// TIA Portal V20 export
FUNCTION "CallDiagnostic" : Void   // FC16, LAD
TITLE = Diagnostics
AUTHOR : SICAR
FAMILY : Diag
// Call of SICAR Diagnostic blocks
// stored: IsIECCheckEnabled true, SetENOAutomatically true
   VAR_TEMP
      statWStringName : WString[24];
      tempHardwareOKexample : Bool;   // REPLACE: This output can be used as an interlock for Control Modules
   END_VAR
   VAR CONSTANT
      TRUE : Bool := TRUE;
   END_VAR
   // Ret_Val : Ret_Val
   VAR_TEMP   // added for the SCL form of the ladder/FBD networks
      _w1 : Bool;
   END_VAR
BEGIN

REGION Network 1: BLOCK INFO HEADER
   // SIEMENS AG / (c)Copyright 2023
   // ------------------------------------------------------------------------------
   // Title:            CallDiagnostic (FC16)
   // Comment/Function: Call of SICAR Diagnostic blocks
   // Library/Family:   Diag
   // Author:           SICAR
   // Tested with:      ---
   // Engineering:      TIA Portal V19
   // Restrictions:     -
   // Requirements:     ---
   // ------------------------------------------------------------------------------
   // Change log table:
   // Version | Date | Expert in charge | Changes applied
   // -------|---------|-------------|--------------------------------------------
   // 01.00.00 | 01.01.1999 | Person x | First released version
   // 01.00.01 | 02.01.1999 | Person y | Block was Updated
END_REGION

REGION Network 2: Call: Diagnostic Profinet Devices
   // For diagnose the whole profinet devices of this PLC
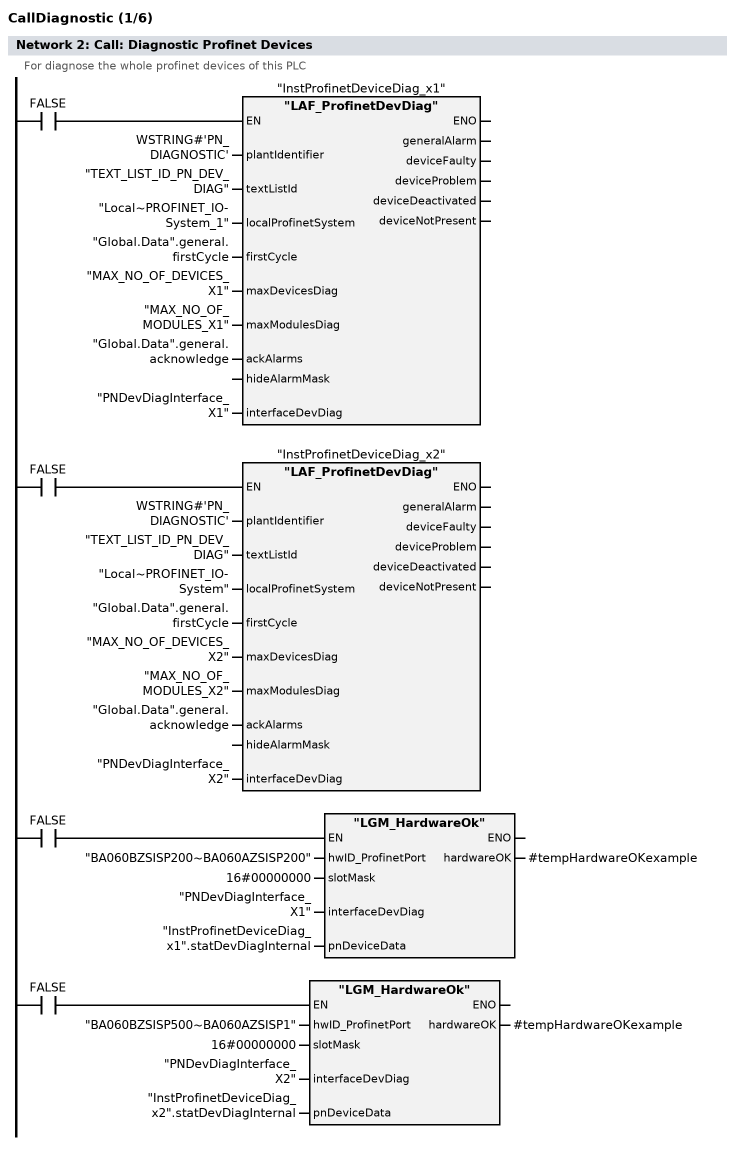
   RUNG wire#powerrail
      Contact( FALSE )
      "InstProfinetDeviceDiag_x1"(plantIdentifier := WSTRING#'PN_DIAGNOSTIC', textListId := "TEXT_LIST_ID_PN_DEV_DIAG", localProfinetSystem := "Local~PROFINET_IO-System_1", firstCycle := "Global.Data".general.firstCycle, maxDevicesDiag := "MAX_NO_OF_DEVICES_X1", maxModulesDiag := "MAX_NO_OF_MODULES_X1", ackAlarms := "Global.Data".general.acknowledge, hideAlarmMask :=, interfaceDevDiag := "PNDevDiagInterface_X1", generalAlarm =>, deviceFaulty =>, deviceProblem =>, deviceDeactivated =>, deviceNotPresent =>)
   END_RUNG
   RUNG wire#powerrail
      Contact( FALSE )
      "InstProfinetDeviceDiag_x2"(plantIdentifier := WSTRING#'PN_DIAGNOSTIC', textListId := "TEXT_LIST_ID_PN_DEV_DIAG", localProfinetSystem := "Local~PROFINET_IO-System", firstCycle := "Global.Data".general.firstCycle, maxDevicesDiag := "MAX_NO_OF_DEVICES_X2", maxModulesDiag := "MAX_NO_OF_MODULES_X2", ackAlarms := "Global.Data".general.acknowledge, hideAlarmMask :=, interfaceDevDiag := "PNDevDiagInterface_X2", generalAlarm =>, deviceFaulty =>, deviceProblem =>, deviceDeactivated =>, deviceNotPresent =>)
   END_RUNG
   RUNG wire#powerrail
      Contact( FALSE )
      "LGM_HardwareOk"(hwID_ProfinetPort := "BA060BZSISP200~BA060AZSISP200", slotMask := 16#00000000, interfaceDevDiag := "PNDevDiagInterface_X1", pnDeviceData := "InstProfinetDeviceDiag_x1".statDevDiagInternal, hardwareOK => #tempHardwareOKexample)
   END_RUNG
   RUNG wire#powerrail
      Contact( FALSE )
      "LGM_HardwareOk"(hwID_ProfinetPort := "BA060BZSISP500~BA060AZSISP1", slotMask := 16#00000000, interfaceDevDiag := "PNDevDiagInterface_X2", pnDeviceData := "InstProfinetDeviceDiag_x2".statDevDiagInternal, hardwareOK => #tempHardwareOKexample)
   END_RUNG
   // the same network as SCL:
   IF FALSE THEN
       "InstProfinetDeviceDiag_x1"(plantIdentifier := WSTRING#'PN_DIAGNOSTIC',   // "LAF_ProfinetDevDiag"
                               textListId := "TEXT_LIST_ID_PN_DEV_DIAG",
                               localProfinetSystem := "Local~PROFINET_IO-System_1",
                               firstCycle := "Global.Data".general.firstCycle,
                               maxDevicesDiag := "MAX_NO_OF_DEVICES_X1",
                               maxModulesDiag := "MAX_NO_OF_MODULES_X1",
                               ackAlarms := "Global.Data".general.acknowledge,
                               interfaceDevDiag := "PNDevDiagInterface_X1");
       "InstProfinetDeviceDiag_x2"(plantIdentifier := WSTRING#'PN_DIAGNOSTIC',   // "LAF_ProfinetDevDiag"
                               textListId := "TEXT_LIST_ID_PN_DEV_DIAG",
                               localProfinetSystem := "Local~PROFINET_IO-System",
                               firstCycle := "Global.Data".general.firstCycle,
                               maxDevicesDiag := "MAX_NO_OF_DEVICES_X2",
                               maxModulesDiag := "MAX_NO_OF_MODULES_X2",
                               ackAlarms := "Global.Data".general.acknowledge,
                               interfaceDevDiag := "PNDevDiagInterface_X2");
       "LGM_HardwareOk"(hwID_ProfinetPort := "BA060BZSISP200~BA060AZSISP200",
                        slotMask := 16#00000000,
                        interfaceDevDiag := "PNDevDiagInterface_X1",
                        pnDeviceData := "InstProfinetDeviceDiag_x1".statDevDiagInternal,
                        hardwareOK => #tempHardwareOKexample);
       "LGM_HardwareOk"(hwID_ProfinetPort := "BA060BZSISP500~BA060AZSISP1",
                        slotMask := 16#00000000,
                        interfaceDevDiag := "PNDevDiagInterface_X2",
                        pnDeviceData := "InstProfinetDeviceDiag_x2".statDevDiagInternal,
                        hardwareOK => #tempHardwareOKexample);
   END_IF;
END_REGION

REGION Network 3: Call: Diagnostic Bool Interface Signals
   // Call the interface bool blocks to show boolean signals on the HMI
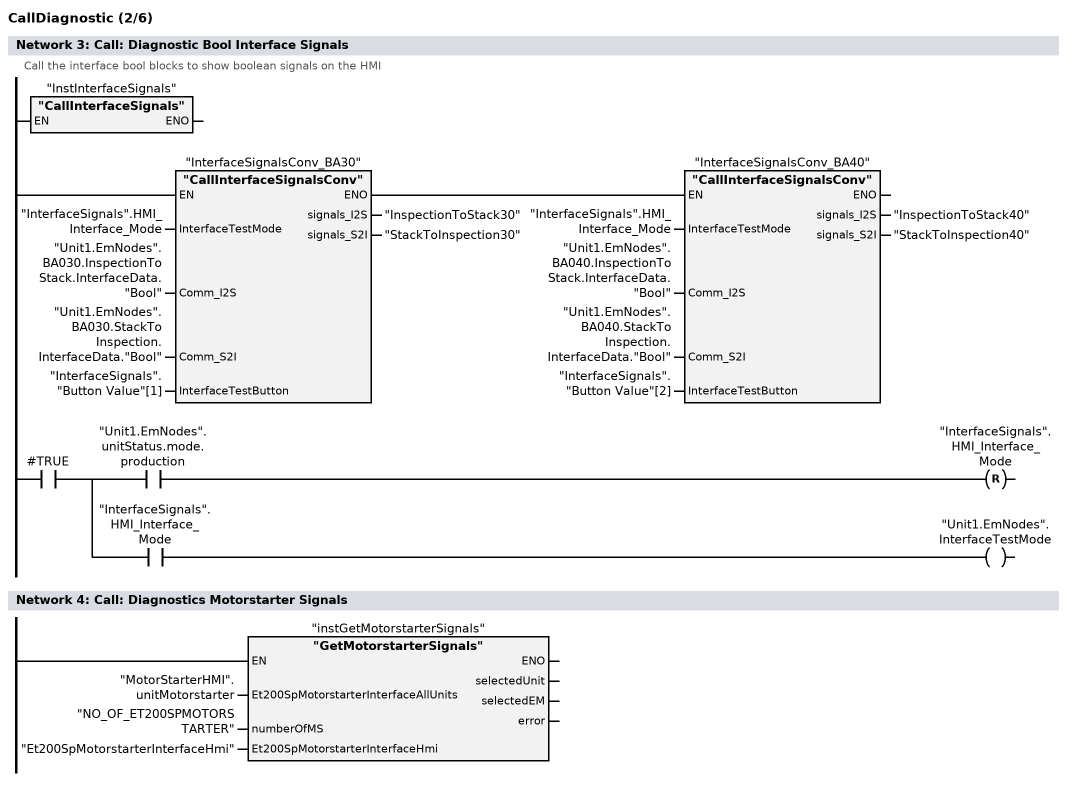
   RUNG wire#powerrail
      "InstInterfaceSignals"()
   END_RUNG
   RUNG wire#powerrail
      "InterfaceSignalsConv_BA30"(InterfaceTestMode := "InterfaceSignals".HMI_Interface_Mode, Comm_I2S := "Unit1.EmNodes".BA030.InspectionToStack.InterfaceData."Bool", Comm_S2I := "Unit1.EmNodes".BA030.StackToInspection.InterfaceData."Bool", InterfaceTestButton := "InterfaceSignals"."Button Value"[1], signals_I2S => "InspectionToStack30", signals_S2I => "StackToInspection30")
      "InterfaceSignalsConv_BA40"(InterfaceTestMode := "InterfaceSignals".HMI_Interface_Mode, Comm_I2S := "Unit1.EmNodes".BA040.InspectionToStack.InterfaceData."Bool", Comm_S2I := "Unit1.EmNodes".BA040.StackToInspection.InterfaceData."Bool", InterfaceTestButton := "InterfaceSignals"."Button Value"[2], signals_I2S => "InspectionToStack40", signals_S2I => "StackToInspection40")
   END_RUNG
   RUNG wire#powerrail
      Contact( #TRUE )
      wire#w1
      Contact( "Unit1.EmNodes".unitStatus.mode.production )
      R_Coil( "InterfaceSignals".HMI_Interface_Mode )
   END_RUNG
   RUNG wire#w1
      Contact( "InterfaceSignals".HMI_Interface_Mode )
      Coil( "Unit1.EmNodes".InterfaceTestMode )
   END_RUNG
   // the same network as SCL:
   "InstInterfaceSignals"();   // "CallInterfaceSignals"
   "InterfaceSignalsConv_BA30"(InterfaceTestMode := "InterfaceSignals".HMI_Interface_Mode,   // "CallInterfaceSignalsConv"
                           Comm_I2S := "Unit1.EmNodes".BA030.InspectionToStack.InterfaceData."Bool",
                           Comm_S2I := "Unit1.EmNodes".BA030.StackToInspection.InterfaceData."Bool",
                           InterfaceTestButton := "InterfaceSignals"."Button Value"[1],
                           signals_I2S => "InspectionToStack30",
                           signals_S2I => "StackToInspection30",
                           ENO => #_w1);
   IF #_w1 THEN
       "InterfaceSignalsConv_BA40"(InterfaceTestMode := "InterfaceSignals".HMI_Interface_Mode,   // "CallInterfaceSignalsConv"
                               Comm_I2S := "Unit1.EmNodes".BA040.InspectionToStack.InterfaceData."Bool",
                               Comm_S2I := "Unit1.EmNodes".BA040.StackToInspection.InterfaceData."Bool",
                               InterfaceTestButton := "InterfaceSignals"."Button Value"[2],
                               signals_I2S => "InspectionToStack40",
                               signals_S2I => "StackToInspection40");
   END_IF;
   IF #TRUE AND "Unit1.EmNodes".unitStatus.mode.production THEN
       "InterfaceSignals".HMI_Interface_Mode := FALSE;
   END_IF;
   "Unit1.EmNodes".InterfaceTestMode := #TRUE AND "InterfaceSignals".HMI_Interface_Mode;
END_REGION

REGION Network 4: Call: Diagnostics Motorstarter Signals
   RUNG wire#powerrail
      "instGetMotorstarterSignals"(Et200SpMotorstarterInterfaceAllUnits := "MotorStarterHMI".unitMotorstarter, numberOfMS := "NO_OF_ET200SPMOTORSTARTER", Et200SpMotorstarterInterfaceHmi := "Et200SpMotorstarterInterfaceHmi", selectedUnit =>, selectedEM =>, error =>)
   END_RUNG
   // the same network as SCL:
   "instGetMotorstarterSignals"(Et200SpMotorstarterInterfaceAllUnits := "MotorStarterHMI".unitMotorstarter,   // "GetMotorstarterSignals"
                           numberOfMS := "NO_OF_ET200SPMOTORSTARTER",
                           Et200SpMotorstarterInterfaceHmi := "Et200SpMotorstarterInterfaceHmi");
END_REGION

REGION Network 5: Call: Diagnostics Drives
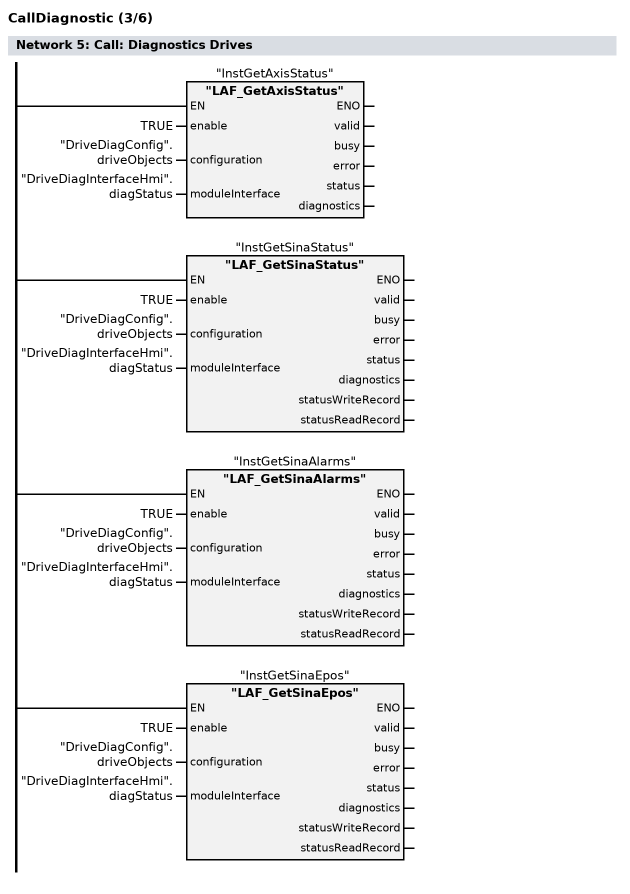
   RUNG wire#powerrail
      "InstGetAxisStatus"(enable := TRUE, configuration := "DriveDiagConfig".driveObjects, moduleInterface := "DriveDiagInterfaceHmi".diagStatus, valid =>, busy =>, error =>, status =>, diagnostics =>)
   END_RUNG
   RUNG wire#powerrail
      "InstGetSinaStatus"(enable := TRUE, configuration := "DriveDiagConfig".driveObjects, moduleInterface := "DriveDiagInterfaceHmi".diagStatus, valid =>, busy =>, error =>, status =>, diagnostics =>, statusWriteRecord =>, statusReadRecord =>)
   END_RUNG
   RUNG wire#powerrail
      "InstGetSinaAlarms"(enable := TRUE, configuration := "DriveDiagConfig".driveObjects, moduleInterface := "DriveDiagInterfaceHmi".diagStatus, valid =>, busy =>, error =>, status =>, diagnostics =>, statusWriteRecord =>, statusReadRecord =>)
   END_RUNG
   RUNG wire#powerrail
      "InstGetSinaEpos"(enable := TRUE, configuration := "DriveDiagConfig".driveObjects, moduleInterface := "DriveDiagInterfaceHmi".diagStatus, valid =>, busy =>, error =>, status =>, diagnostics =>, statusWriteRecord =>, statusReadRecord =>)
   END_RUNG
   // the same network as SCL:
   "InstGetAxisStatus"(enable := TRUE,   // "LAF_GetAxisStatus"
                       configuration := "DriveDiagConfig".driveObjects,
                       moduleInterface := "DriveDiagInterfaceHmi".diagStatus);
   "InstGetSinaStatus"(enable := TRUE,   // "LAF_GetSinaStatus"
                       configuration := "DriveDiagConfig".driveObjects,
                       moduleInterface := "DriveDiagInterfaceHmi".diagStatus);
   "InstGetSinaAlarms"(enable := TRUE,   // "LAF_GetSinaAlarms"
                       configuration := "DriveDiagConfig".driveObjects,
                       moduleInterface := "DriveDiagInterfaceHmi".diagStatus);
   "InstGetSinaEpos"(enable := TRUE,   // "LAF_GetSinaEpos"
                     configuration := "DriveDiagConfig".driveObjects,
                     moduleInterface := "DriveDiagInterfaceHmi".diagStatus);
END_REGION

REGION Network 6: Call: Servo Torque Cal (DR1~10)
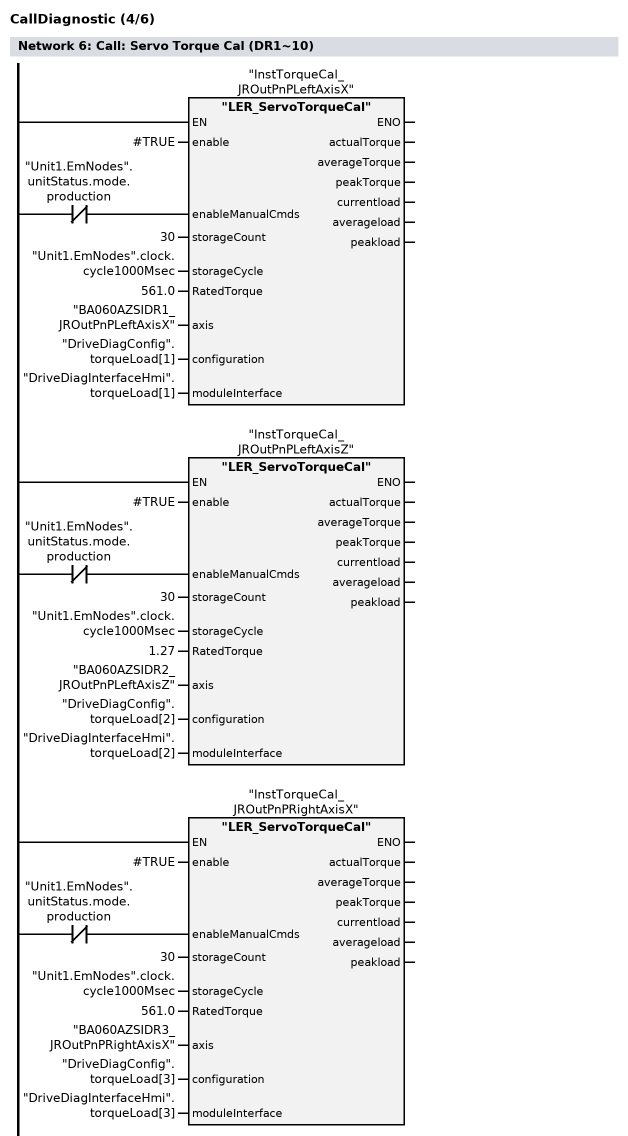
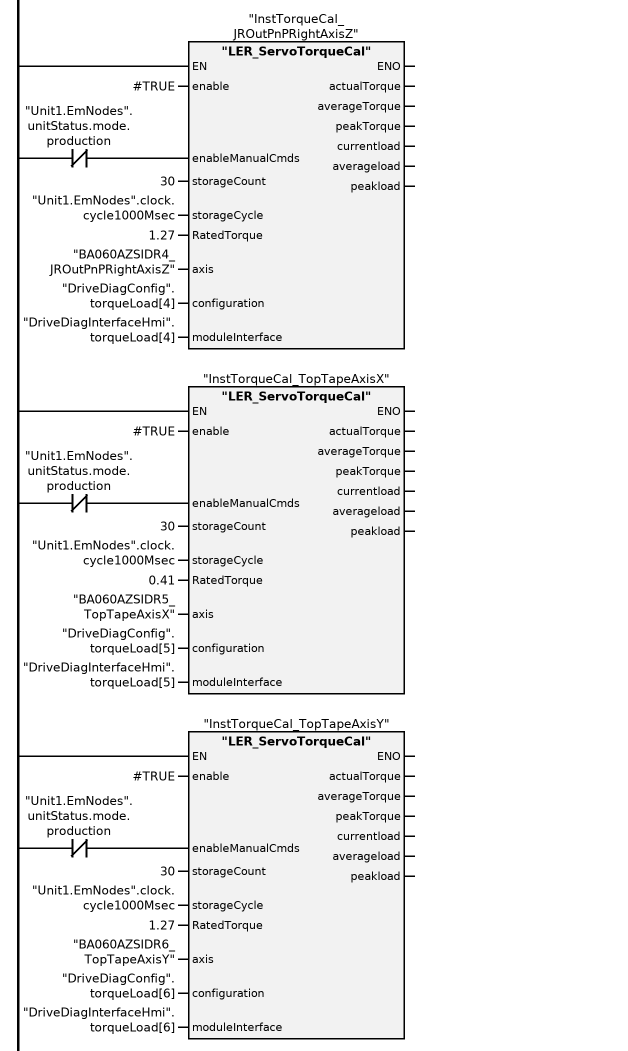
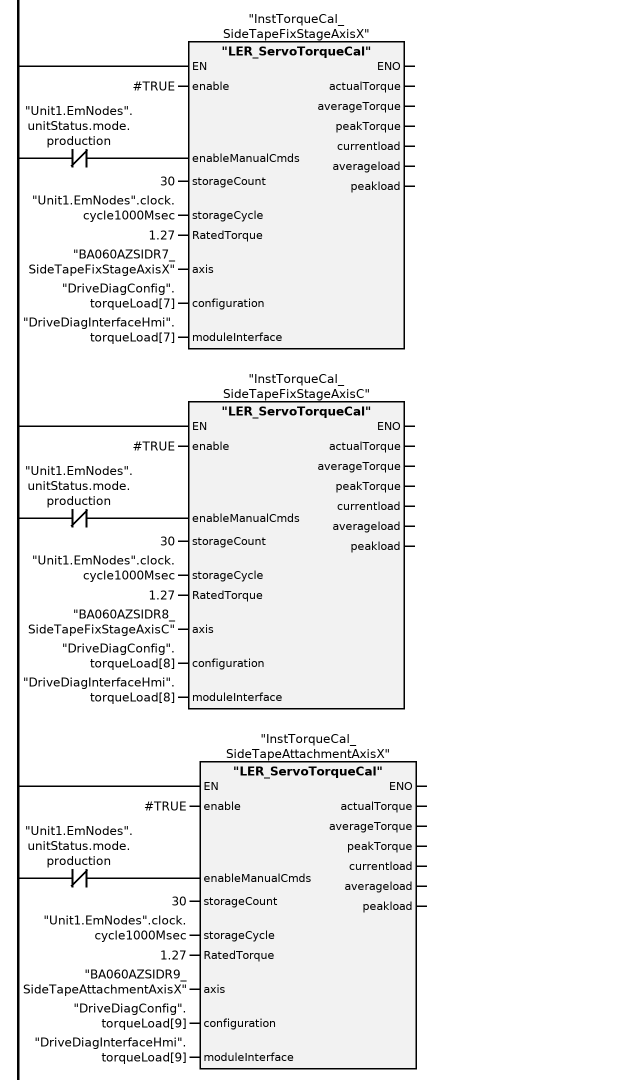
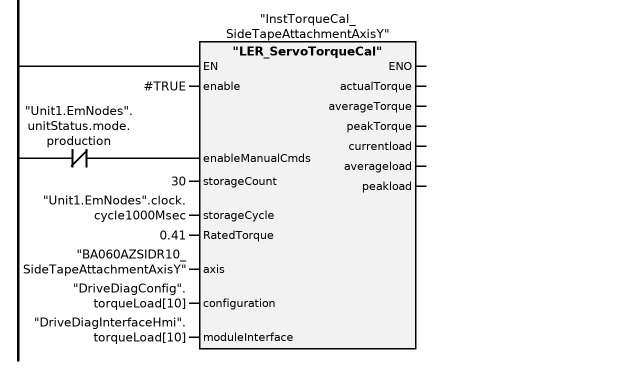
   RUNG wire#powerrail
      "InstTorqueCal_JROutPnPLeftAxisX"(enableManualCmds := wire#w1, enable := #TRUE, storageCount := 30, storageCycle := "Unit1.EmNodes".clock.cycle1000Msec, RatedTorque := 561.0, axis := "BA060AZSIDR1_JROutPnPLeftAxisX", configuration := "DriveDiagConfig".torqueLoad[1], moduleInterface := "DriveDiagInterfaceHmi".torqueLoad[1], actualTorque =>, averageTorque =>, peakTorque =>, currentload =>, averageload =>, peakload =>)
   END_RUNG
   RUNG wire#powerrail
      I_Contact( "Unit1.EmNodes".unitStatus.mode.production )
   END_RUNG wire#w1
   RUNG wire#powerrail
      "InstTorqueCal_JROutPnPLeftAxisZ"(enableManualCmds := wire#w2, enable := #TRUE, storageCount := 30, storageCycle := "Unit1.EmNodes".clock.cycle1000Msec, RatedTorque := 1.27, axis := "BA060AZSIDR2_JROutPnPLeftAxisZ", configuration := "DriveDiagConfig".torqueLoad[2], moduleInterface := "DriveDiagInterfaceHmi".torqueLoad[2], actualTorque =>, averageTorque =>, peakTorque =>, currentload =>, averageload =>, peakload =>)
   END_RUNG
   RUNG wire#powerrail
      I_Contact( "Unit1.EmNodes".unitStatus.mode.production )
   END_RUNG wire#w2
   RUNG wire#powerrail
      "InstTorqueCal_JROutPnPRightAxisX"(enableManualCmds := wire#w3, enable := #TRUE, storageCount := 30, storageCycle := "Unit1.EmNodes".clock.cycle1000Msec, RatedTorque := 561.0, axis := "BA060AZSIDR3_JROutPnPRightAxisX", configuration := "DriveDiagConfig".torqueLoad[3], moduleInterface := "DriveDiagInterfaceHmi".torqueLoad[3], actualTorque =>, averageTorque =>, peakTorque =>, currentload =>, averageload =>, peakload =>)
   END_RUNG
   RUNG wire#powerrail
      I_Contact( "Unit1.EmNodes".unitStatus.mode.production )
   END_RUNG wire#w3
   RUNG wire#powerrail
      "InstTorqueCal_JROutPnPRightAxisZ"(enableManualCmds := wire#w4, enable := #TRUE, storageCount := 30, storageCycle := "Unit1.EmNodes".clock.cycle1000Msec, RatedTorque := 1.27, axis := "BA060AZSIDR4_JROutPnPRightAxisZ", configuration := "DriveDiagConfig".torqueLoad[4], moduleInterface := "DriveDiagInterfaceHmi".torqueLoad[4], actualTorque =>, averageTorque =>, peakTorque =>, currentload =>, averageload =>, peakload =>)
   END_RUNG
   RUNG wire#powerrail
      I_Contact( "Unit1.EmNodes".unitStatus.mode.production )
   END_RUNG wire#w4
   RUNG wire#powerrail
      "InstTorqueCal_TopTapeAxisX"(enableManualCmds := wire#w5, enable := #TRUE, storageCount := 30, storageCycle := "Unit1.EmNodes".clock.cycle1000Msec, RatedTorque := 0.41, axis := "BA060AZSIDR5_TopTapeAxisX", configuration := "DriveDiagConfig".torqueLoad[5], moduleInterface := "DriveDiagInterfaceHmi".torqueLoad[5], actualTorque =>, averageTorque =>, peakTorque =>, currentload =>, averageload =>, peakload =>)
   END_RUNG
   RUNG wire#powerrail
      I_Contact( "Unit1.EmNodes".unitStatus.mode.production )
   END_RUNG wire#w5
   RUNG wire#powerrail
      "InstTorqueCal_TopTapeAxisY"(enableManualCmds := wire#w6, enable := #TRUE, storageCount := 30, storageCycle := "Unit1.EmNodes".clock.cycle1000Msec, RatedTorque := 1.27, axis := "BA060AZSIDR6_TopTapeAxisY", configuration := "DriveDiagConfig".torqueLoad[6], moduleInterface := "DriveDiagInterfaceHmi".torqueLoad[6], actualTorque =>, averageTorque =>, peakTorque =>, currentload =>, averageload =>, peakload =>)
   END_RUNG
   RUNG wire#powerrail
      I_Contact( "Unit1.EmNodes".unitStatus.mode.production )
   END_RUNG wire#w6
   RUNG wire#powerrail
      "InstTorqueCal_SideTapeFixStageAxisX"(enableManualCmds := wire#w7, enable := #TRUE, storageCount := 30, storageCycle := "Unit1.EmNodes".clock.cycle1000Msec, RatedTorque := 1.27, axis := "BA060AZSIDR7_SideTapeFixStageAxisX", configuration := "DriveDiagConfig".torqueLoad[7], moduleInterface := "DriveDiagInterfaceHmi".torqueLoad[7], actualTorque =>, averageTorque =>, peakTorque =>, currentload =>, averageload =>, peakload =>)
   END_RUNG
   RUNG wire#powerrail
      I_Contact( "Unit1.EmNodes".unitStatus.mode.production )
   END_RUNG wire#w7
   RUNG wire#powerrail
      "InstTorqueCal_SideTapeFixStageAxisC"(enableManualCmds := wire#w8, enable := #TRUE, storageCount := 30, storageCycle := "Unit1.EmNodes".clock.cycle1000Msec, RatedTorque := 1.27, axis := "BA060AZSIDR8_SideTapeFixStageAxisC", configuration := "DriveDiagConfig".torqueLoad[8], moduleInterface := "DriveDiagInterfaceHmi".torqueLoad[8], actualTorque =>, averageTorque =>, peakTorque =>, currentload =>, averageload =>, peakload =>)
   END_RUNG
   RUNG wire#powerrail
      I_Contact( "Unit1.EmNodes".unitStatus.mode.production )
   END_RUNG wire#w8
   RUNG wire#powerrail
      "InstTorqueCal_SideTapeAttachmentAxisX"(enableManualCmds := wire#w9, enable := #TRUE, storageCount := 30, storageCycle := "Unit1.EmNodes".clock.cycle1000Msec, RatedTorque := 1.27, axis := "BA060AZSIDR9_SideTapeAttachmentAxisX", configuration := "DriveDiagConfig".torqueLoad[9], moduleInterface := "DriveDiagInterfaceHmi".torqueLoad[9], actualTorque =>, averageTorque =>, peakTorque =>, currentload =>, averageload =>, peakload =>)
   END_RUNG
   RUNG wire#powerrail
      I_Contact( "Unit1.EmNodes".unitStatus.mode.production )
   END_RUNG wire#w9
   RUNG wire#powerrail
      "InstTorqueCal_SideTapeAttachmentAxisY"(enableManualCmds := wire#w10, enable := #TRUE, storageCount := 30, storageCycle := "Unit1.EmNodes".clock.cycle1000Msec, RatedTorque := 0.41, axis := "BA060AZSIDR10_SideTapeAttachmentAxisY", configuration := "DriveDiagConfig".torqueLoad[10], moduleInterface := "DriveDiagInterfaceHmi".torqueLoad[10], actualTorque =>, averageTorque =>, peakTorque =>, currentload =>, averageload =>, peakload =>)
   END_RUNG
   RUNG wire#powerrail
      I_Contact( "Unit1.EmNodes".unitStatus.mode.production )
   END_RUNG wire#w10
   // the same network as SCL:
   "InstTorqueCal_JROutPnPLeftAxisX"(enable := #TRUE,   // "LER_ServoTorqueCal"
                           enableManualCmds := NOT "Unit1.EmNodes".unitStatus.mode.production,
                           storageCount := 30,
                           storageCycle := "Unit1.EmNodes".clock.cycle1000Msec,
                           RatedTorque := 561.0,
                           axis := "BA060AZSIDR1_JROutPnPLeftAxisX",
                           configuration := "DriveDiagConfig".torqueLoad[1],
                           moduleInterface := "DriveDiagInterfaceHmi".torqueLoad[1]);
   "InstTorqueCal_JROutPnPLeftAxisZ"(enable := #TRUE,   // "LER_ServoTorqueCal"
                           enableManualCmds := NOT "Unit1.EmNodes".unitStatus.mode.production,
                           storageCount := 30,
                           storageCycle := "Unit1.EmNodes".clock.cycle1000Msec,
                           RatedTorque := 1.27,
                           axis := "BA060AZSIDR2_JROutPnPLeftAxisZ",
                           configuration := "DriveDiagConfig".torqueLoad[2],
                           moduleInterface := "DriveDiagInterfaceHmi".torqueLoad[2]);
   "InstTorqueCal_JROutPnPRightAxisX"(enable := #TRUE,   // "LER_ServoTorqueCal"
                           enableManualCmds := NOT "Unit1.EmNodes".unitStatus.mode.production,
                           storageCount := 30,
                           storageCycle := "Unit1.EmNodes".clock.cycle1000Msec,
                           RatedTorque := 561.0,
                           axis := "BA060AZSIDR3_JROutPnPRightAxisX",
                           configuration := "DriveDiagConfig".torqueLoad[3],
                           moduleInterface := "DriveDiagInterfaceHmi".torqueLoad[3]);
   "InstTorqueCal_JROutPnPRightAxisZ"(enable := #TRUE,   // "LER_ServoTorqueCal"
                           enableManualCmds := NOT "Unit1.EmNodes".unitStatus.mode.production,
                           storageCount := 30,
                           storageCycle := "Unit1.EmNodes".clock.cycle1000Msec,
                           RatedTorque := 1.27,
                           axis := "BA060AZSIDR4_JROutPnPRightAxisZ",
                           configuration := "DriveDiagConfig".torqueLoad[4],
                           moduleInterface := "DriveDiagInterfaceHmi".torqueLoad[4]);
   "InstTorqueCal_TopTapeAxisX"(enable := #TRUE,   // "LER_ServoTorqueCal"
                           enableManualCmds := NOT "Unit1.EmNodes".unitStatus.mode.production,
                           storageCount := 30,
                           storageCycle := "Unit1.EmNodes".clock.cycle1000Msec,
                           RatedTorque := 0.41,
                           axis := "BA060AZSIDR5_TopTapeAxisX",
                           configuration := "DriveDiagConfig".torqueLoad[5],
                           moduleInterface := "DriveDiagInterfaceHmi".torqueLoad[5]);
   "InstTorqueCal_TopTapeAxisY"(enable := #TRUE,   // "LER_ServoTorqueCal"
                           enableManualCmds := NOT "Unit1.EmNodes".unitStatus.mode.production,
                           storageCount := 30,
                           storageCycle := "Unit1.EmNodes".clock.cycle1000Msec,
                           RatedTorque := 1.27,
                           axis := "BA060AZSIDR6_TopTapeAxisY",
                           configuration := "DriveDiagConfig".torqueLoad[6],
                           moduleInterface := "DriveDiagInterfaceHmi".torqueLoad[6]);
   "InstTorqueCal_SideTapeFixStageAxisX"(enable := #TRUE,   // "LER_ServoTorqueCal"
                           enableManualCmds := NOT "Unit1.EmNodes".unitStatus.mode.production,
                           storageCount := 30,
                           storageCycle := "Unit1.EmNodes".clock.cycle1000Msec,
                           RatedTorque := 1.27,
                           axis := "BA060AZSIDR7_SideTapeFixStageAxisX",
                           configuration := "DriveDiagConfig".torqueLoad[7],
                           moduleInterface := "DriveDiagInterfaceHmi".torqueLoad[7]);
   "InstTorqueCal_SideTapeFixStageAxisC"(enable := #TRUE,   // "LER_ServoTorqueCal"
                           enableManualCmds := NOT "Unit1.EmNodes".unitStatus.mode.production,
                           storageCount := 30,
                           storageCycle := "Unit1.EmNodes".clock.cycle1000Msec,
                           RatedTorque := 1.27,
                           axis := "BA060AZSIDR8_SideTapeFixStageAxisC",
                           configuration := "DriveDiagConfig".torqueLoad[8],
                           moduleInterface := "DriveDiagInterfaceHmi".torqueLoad[8]);
   "InstTorqueCal_SideTapeAttachmentAxisX"(enable := #TRUE,   // "LER_ServoTorqueCal"
                           enableManualCmds := NOT "Unit1.EmNodes".unitStatus.mode.production,
                           storageCount := 30,
                           storageCycle := "Unit1.EmNodes".clock.cycle1000Msec,
                           RatedTorque := 1.27,
                           axis := "BA060AZSIDR9_SideTapeAttachmentAxisX",
                           configuration := "DriveDiagConfig".torqueLoad[9],
                           moduleInterface := "DriveDiagInterfaceHmi".torqueLoad[9]);
   "InstTorqueCal_SideTapeAttachmentAxisY"(enable := #TRUE,   // "LER_ServoTorqueCal"
                           enableManualCmds := NOT "Unit1.EmNodes".unitStatus.mode.production,
                           storageCount := 30,
                           storageCycle := "Unit1.EmNodes".clock.cycle1000Msec,
                           RatedTorque := 0.41,
                           axis := "BA060AZSIDR10_SideTapeAttachmentAxisY",
                           configuration := "DriveDiagConfig".torqueLoad[10],
                           moduleInterface := "DriveDiagInterfaceHmi".torqueLoad[10]);
END_REGION

REGION Network 7: Call: Servo Torque Cal (DR11~20)
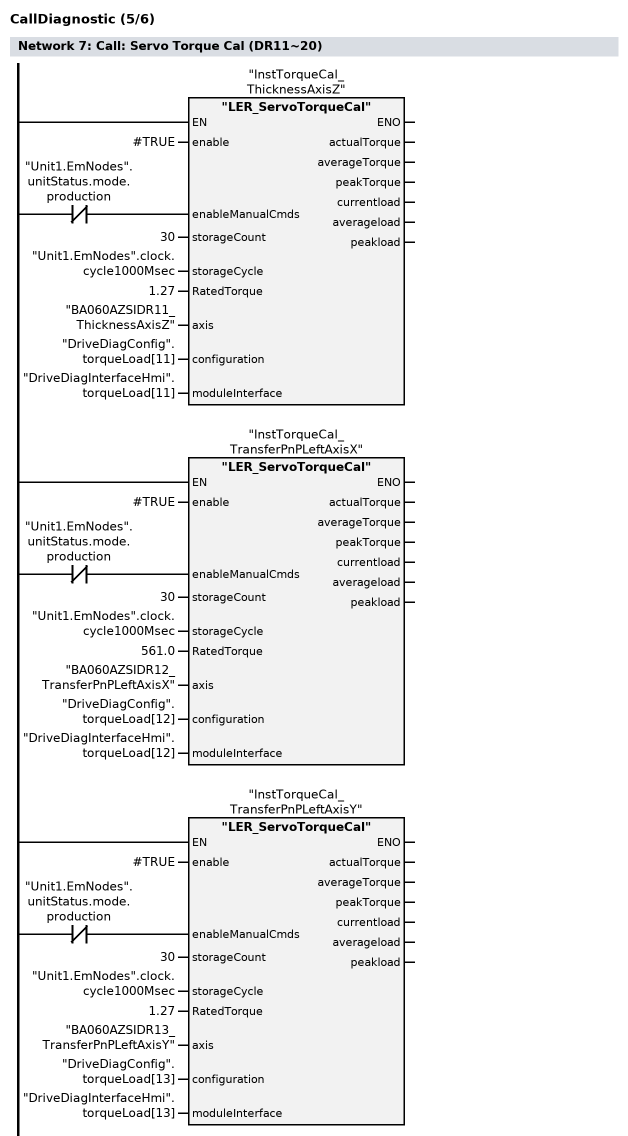
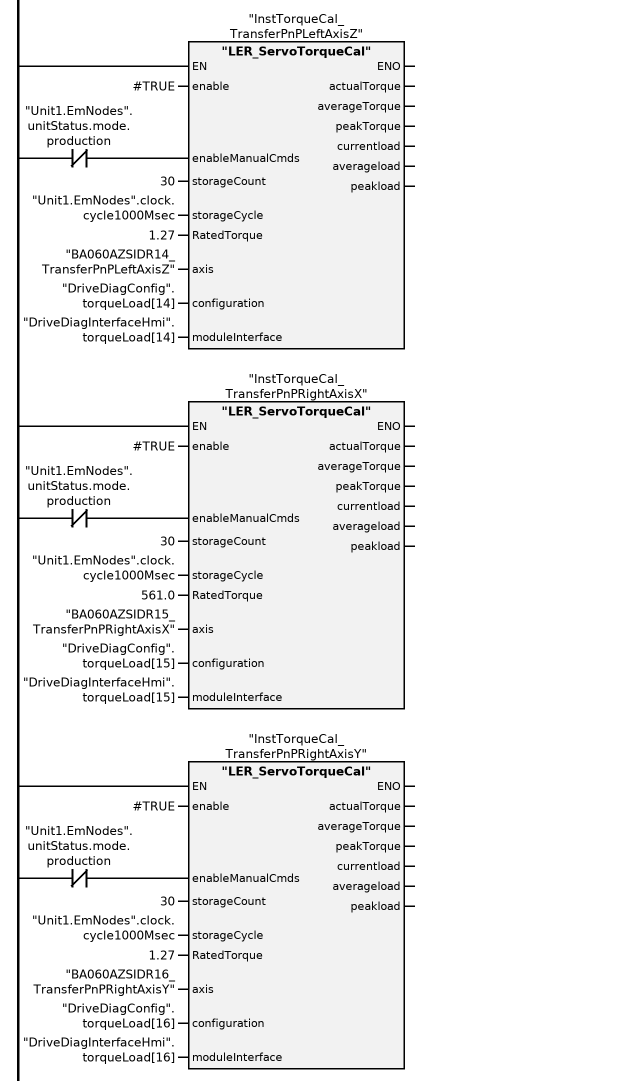
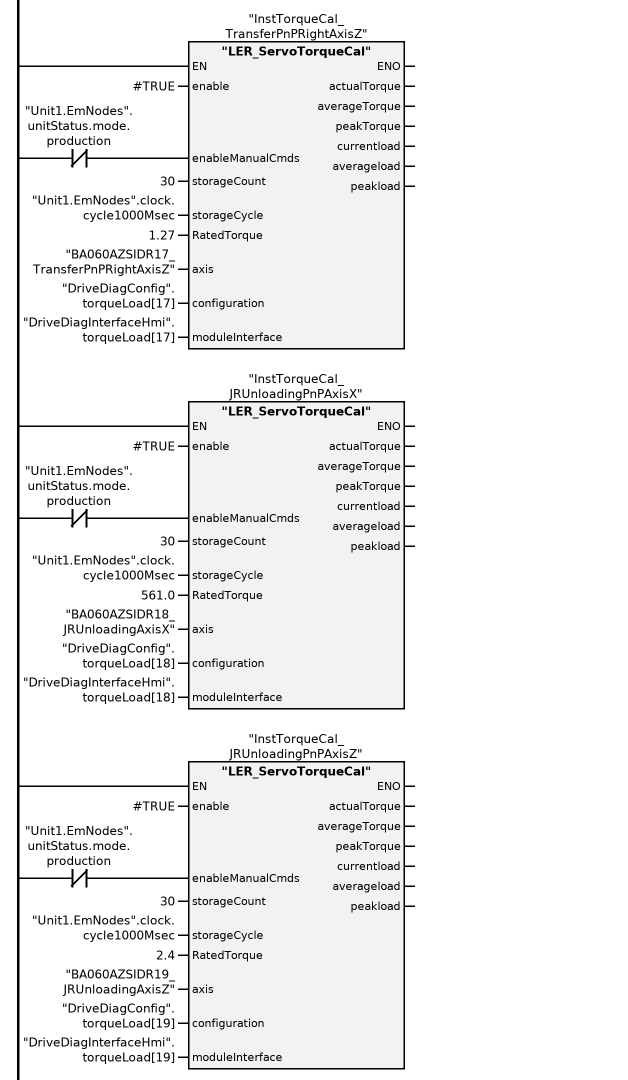
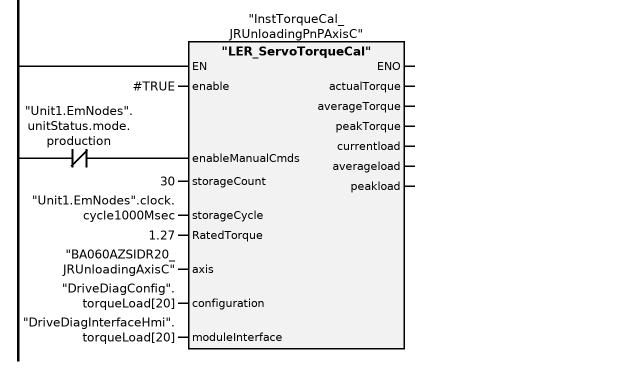
   RUNG wire#powerrail
      "InstTorqueCal_ThicknessAxisZ"(enableManualCmds := wire#w1, enable := #TRUE, storageCount := 30, storageCycle := "Unit1.EmNodes".clock.cycle1000Msec, RatedTorque := 1.27, axis := "BA060AZSIDR11_ThicknessAxisZ", configuration := "DriveDiagConfig".torqueLoad[11], moduleInterface := "DriveDiagInterfaceHmi".torqueLoad[11], actualTorque =>, averageTorque =>, peakTorque =>, currentload =>, averageload =>, peakload =>)
   END_RUNG
   RUNG wire#powerrail
      I_Contact( "Unit1.EmNodes".unitStatus.mode.production )
   END_RUNG wire#w1
   RUNG wire#powerrail
      "InstTorqueCal_TransferPnPLeftAxisX"(enableManualCmds := wire#w2, enable := #TRUE, storageCount := 30, storageCycle := "Unit1.EmNodes".clock.cycle1000Msec, RatedTorque := 561.0, axis := "BA060AZSIDR12_TransferPnPLeftAxisX", configuration := "DriveDiagConfig".torqueLoad[12], moduleInterface := "DriveDiagInterfaceHmi".torqueLoad[12], actualTorque =>, averageTorque =>, peakTorque =>, currentload =>, averageload =>, peakload =>)
   END_RUNG
   RUNG wire#powerrail
      I_Contact( "Unit1.EmNodes".unitStatus.mode.production )
   END_RUNG wire#w2
   RUNG wire#powerrail
      "InstTorqueCal_TransferPnPLeftAxisY"(enableManualCmds := wire#w3, enable := #TRUE, storageCount := 30, storageCycle := "Unit1.EmNodes".clock.cycle1000Msec, RatedTorque := 1.27, axis := "BA060AZSIDR13_TransferPnPLeftAxisY", configuration := "DriveDiagConfig".torqueLoad[13], moduleInterface := "DriveDiagInterfaceHmi".torqueLoad[13], actualTorque =>, averageTorque =>, peakTorque =>, currentload =>, averageload =>, peakload =>)
   END_RUNG
   RUNG wire#powerrail
      I_Contact( "Unit1.EmNodes".unitStatus.mode.production )
   END_RUNG wire#w3
   RUNG wire#powerrail
      "InstTorqueCal_TransferPnPLeftAxisZ"(enableManualCmds := wire#w4, enable := #TRUE, storageCount := 30, storageCycle := "Unit1.EmNodes".clock.cycle1000Msec, RatedTorque := 1.27, axis := "BA060AZSIDR14_TransferPnPLeftAxisZ", configuration := "DriveDiagConfig".torqueLoad[14], moduleInterface := "DriveDiagInterfaceHmi".torqueLoad[14], actualTorque =>, averageTorque =>, peakTorque =>, currentload =>, averageload =>, peakload =>)
   END_RUNG
   RUNG wire#powerrail
      I_Contact( "Unit1.EmNodes".unitStatus.mode.production )
   END_RUNG wire#w4
   RUNG wire#powerrail
      "InstTorqueCal_TransferPnPRightAxisX"(enableManualCmds := wire#w5, enable := #TRUE, storageCount := 30, storageCycle := "Unit1.EmNodes".clock.cycle1000Msec, RatedTorque := 561.0, axis := "BA060AZSIDR15_TransferPnPRightAxisX", configuration := "DriveDiagConfig".torqueLoad[15], moduleInterface := "DriveDiagInterfaceHmi".torqueLoad[15], actualTorque =>, averageTorque =>, peakTorque =>, currentload =>, averageload =>, peakload =>)
   END_RUNG
   RUNG wire#powerrail
      I_Contact( "Unit1.EmNodes".unitStatus.mode.production )
   END_RUNG wire#w5
   RUNG wire#powerrail
      "InstTorqueCal_TransferPnPRightAxisY"(enableManualCmds := wire#w6, enable := #TRUE, storageCount := 30, storageCycle := "Unit1.EmNodes".clock.cycle1000Msec, RatedTorque := 1.27, axis := "BA060AZSIDR16_TransferPnPRightAxisY", configuration := "DriveDiagConfig".torqueLoad[16], moduleInterface := "DriveDiagInterfaceHmi".torqueLoad[16], actualTorque =>, averageTorque =>, peakTorque =>, currentload =>, averageload =>, peakload =>)
   END_RUNG
   RUNG wire#powerrail
      I_Contact( "Unit1.EmNodes".unitStatus.mode.production )
   END_RUNG wire#w6
   RUNG wire#powerrail
      "InstTorqueCal_TransferPnPRightAxisZ"(enableManualCmds := wire#w7, enable := #TRUE, storageCount := 30, storageCycle := "Unit1.EmNodes".clock.cycle1000Msec, RatedTorque := 1.27, axis := "BA060AZSIDR17_TransferPnPRightAxisZ", configuration := "DriveDiagConfig".torqueLoad[17], moduleInterface := "DriveDiagInterfaceHmi".torqueLoad[17], actualTorque =>, averageTorque =>, peakTorque =>, currentload =>, averageload =>, peakload =>)
   END_RUNG
   RUNG wire#powerrail
      I_Contact( "Unit1.EmNodes".unitStatus.mode.production )
   END_RUNG wire#w7
   RUNG wire#powerrail
      "InstTorqueCal_JRUnloadingPnPAxisX"(enableManualCmds := wire#w8, enable := #TRUE, storageCount := 30, storageCycle := "Unit1.EmNodes".clock.cycle1000Msec, RatedTorque := 561.0, axis := "BA060AZSIDR18_JRUnloadingAxisX", configuration := "DriveDiagConfig".torqueLoad[18], moduleInterface := "DriveDiagInterfaceHmi".torqueLoad[18], actualTorque =>, averageTorque =>, peakTorque =>, currentload =>, averageload =>, peakload =>)
   END_RUNG
   RUNG wire#powerrail
      I_Contact( "Unit1.EmNodes".unitStatus.mode.production )
   END_RUNG wire#w8
   RUNG wire#powerrail
      "InstTorqueCal_JRUnloadingPnPAxisZ"(enableManualCmds := wire#w9, enable := #TRUE, storageCount := 30, storageCycle := "Unit1.EmNodes".clock.cycle1000Msec, RatedTorque := 2.4, axis := "BA060AZSIDR19_JRUnloadingAxisZ", configuration := "DriveDiagConfig".torqueLoad[19], moduleInterface := "DriveDiagInterfaceHmi".torqueLoad[19], actualTorque =>, averageTorque =>, peakTorque =>, currentload =>, averageload =>, peakload =>)
   END_RUNG
   RUNG wire#powerrail
      I_Contact( "Unit1.EmNodes".unitStatus.mode.production )
   END_RUNG wire#w9
   RUNG wire#powerrail
      "InstTorqueCal_JRUnloadingPnPAxisC"(enableManualCmds := wire#w10, enable := #TRUE, storageCount := 30, storageCycle := "Unit1.EmNodes".clock.cycle1000Msec, RatedTorque := 1.27, axis := "BA060AZSIDR20_JRUnloadingAxisC", configuration := "DriveDiagConfig".torqueLoad[20], moduleInterface := "DriveDiagInterfaceHmi".torqueLoad[20], actualTorque =>, averageTorque =>, peakTorque =>, currentload =>, averageload =>, peakload =>)
   END_RUNG
   RUNG wire#powerrail
      I_Contact( "Unit1.EmNodes".unitStatus.mode.production )
   END_RUNG wire#w10
   // the same network as SCL:
   "InstTorqueCal_ThicknessAxisZ"(enable := #TRUE,   // "LER_ServoTorqueCal"
                           enableManualCmds := NOT "Unit1.EmNodes".unitStatus.mode.production,
                           storageCount := 30,
                           storageCycle := "Unit1.EmNodes".clock.cycle1000Msec,
                           RatedTorque := 1.27,
                           axis := "BA060AZSIDR11_ThicknessAxisZ",
                           configuration := "DriveDiagConfig".torqueLoad[11],
                           moduleInterface := "DriveDiagInterfaceHmi".torqueLoad[11]);
   "InstTorqueCal_TransferPnPLeftAxisX"(enable := #TRUE,   // "LER_ServoTorqueCal"
                           enableManualCmds := NOT "Unit1.EmNodes".unitStatus.mode.production,
                           storageCount := 30,
                           storageCycle := "Unit1.EmNodes".clock.cycle1000Msec,
                           RatedTorque := 561.0,
                           axis := "BA060AZSIDR12_TransferPnPLeftAxisX",
                           configuration := "DriveDiagConfig".torqueLoad[12],
                           moduleInterface := "DriveDiagInterfaceHmi".torqueLoad[12]);
   "InstTorqueCal_TransferPnPLeftAxisY"(enable := #TRUE,   // "LER_ServoTorqueCal"
                           enableManualCmds := NOT "Unit1.EmNodes".unitStatus.mode.production,
                           storageCount := 30,
                           storageCycle := "Unit1.EmNodes".clock.cycle1000Msec,
                           RatedTorque := 1.27,
                           axis := "BA060AZSIDR13_TransferPnPLeftAxisY",
                           configuration := "DriveDiagConfig".torqueLoad[13],
                           moduleInterface := "DriveDiagInterfaceHmi".torqueLoad[13]);
   "InstTorqueCal_TransferPnPLeftAxisZ"(enable := #TRUE,   // "LER_ServoTorqueCal"
                           enableManualCmds := NOT "Unit1.EmNodes".unitStatus.mode.production,
                           storageCount := 30,
                           storageCycle := "Unit1.EmNodes".clock.cycle1000Msec,
                           RatedTorque := 1.27,
                           axis := "BA060AZSIDR14_TransferPnPLeftAxisZ",
                           configuration := "DriveDiagConfig".torqueLoad[14],
                           moduleInterface := "DriveDiagInterfaceHmi".torqueLoad[14]);
   "InstTorqueCal_TransferPnPRightAxisX"(enable := #TRUE,   // "LER_ServoTorqueCal"
                           enableManualCmds := NOT "Unit1.EmNodes".unitStatus.mode.production,
                           storageCount := 30,
                           storageCycle := "Unit1.EmNodes".clock.cycle1000Msec,
                           RatedTorque := 561.0,
                           axis := "BA060AZSIDR15_TransferPnPRightAxisX",
                           configuration := "DriveDiagConfig".torqueLoad[15],
                           moduleInterface := "DriveDiagInterfaceHmi".torqueLoad[15]);
   "InstTorqueCal_TransferPnPRightAxisY"(enable := #TRUE,   // "LER_ServoTorqueCal"
                           enableManualCmds := NOT "Unit1.EmNodes".unitStatus.mode.production,
                           storageCount := 30,
                           storageCycle := "Unit1.EmNodes".clock.cycle1000Msec,
                           RatedTorque := 1.27,
                           axis := "BA060AZSIDR16_TransferPnPRightAxisY",
                           configuration := "DriveDiagConfig".torqueLoad[16],
                           moduleInterface := "DriveDiagInterfaceHmi".torqueLoad[16]);
   "InstTorqueCal_TransferPnPRightAxisZ"(enable := #TRUE,   // "LER_ServoTorqueCal"
                           enableManualCmds := NOT "Unit1.EmNodes".unitStatus.mode.production,
                           storageCount := 30,
                           storageCycle := "Unit1.EmNodes".clock.cycle1000Msec,
                           RatedTorque := 1.27,
                           axis := "BA060AZSIDR17_TransferPnPRightAxisZ",
                           configuration := "DriveDiagConfig".torqueLoad[17],
                           moduleInterface := "DriveDiagInterfaceHmi".torqueLoad[17]);
   "InstTorqueCal_JRUnloadingPnPAxisX"(enable := #TRUE,   // "LER_ServoTorqueCal"
                           enableManualCmds := NOT "Unit1.EmNodes".unitStatus.mode.production,
                           storageCount := 30,
                           storageCycle := "Unit1.EmNodes".clock.cycle1000Msec,
                           RatedTorque := 561.0,
                           axis := "BA060AZSIDR18_JRUnloadingAxisX",
                           configuration := "DriveDiagConfig".torqueLoad[18],
                           moduleInterface := "DriveDiagInterfaceHmi".torqueLoad[18]);
   "InstTorqueCal_JRUnloadingPnPAxisZ"(enable := #TRUE,   // "LER_ServoTorqueCal"
                           enableManualCmds := NOT "Unit1.EmNodes".unitStatus.mode.production,
                           storageCount := 30,
                           storageCycle := "Unit1.EmNodes".clock.cycle1000Msec,
                           RatedTorque := 2.4,
                           axis := "BA060AZSIDR19_JRUnloadingAxisZ",
                           configuration := "DriveDiagConfig".torqueLoad[19],
                           moduleInterface := "DriveDiagInterfaceHmi".torqueLoad[19]);
   "InstTorqueCal_JRUnloadingPnPAxisC"(enable := #TRUE,   // "LER_ServoTorqueCal"
                           enableManualCmds := NOT "Unit1.EmNodes".unitStatus.mode.production,
                           storageCount := 30,
                           storageCycle := "Unit1.EmNodes".clock.cycle1000Msec,
                           RatedTorque := 1.27,
                           axis := "BA060AZSIDR20_JRUnloadingAxisC",
                           configuration := "DriveDiagConfig".torqueLoad[20],
                           moduleInterface := "DriveDiagInterfaceHmi".torqueLoad[20]);
END_REGION

REGION Network 8: Call RFID simulation
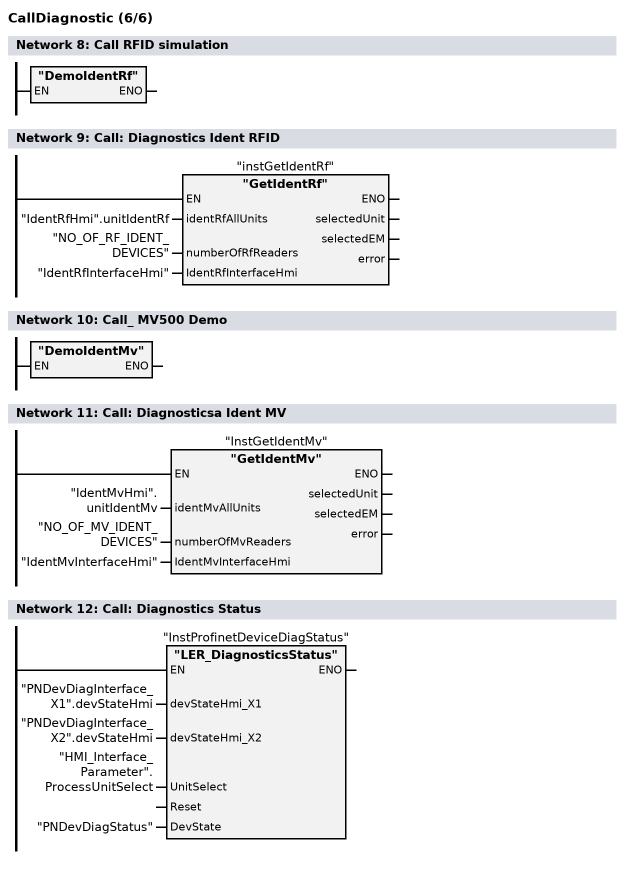
   RUNG wire#powerrail
      "DemoIdentRf"()
   END_RUNG
   // the same network as SCL:
   "DemoIdentRf"();
END_REGION

REGION Network 9: Call: Diagnostics Ident RFID
   RUNG wire#powerrail
      "instGetIdentRf"(identRfAllUnits := "IdentRfHmi".unitIdentRf, numberOfRfReaders := "NO_OF_RF_IDENT_DEVICES", IdentRfInterfaceHmi := "IdentRfInterfaceHmi", selectedUnit =>, selectedEM =>, error =>)
   END_RUNG
   // the same network as SCL:
   "instGetIdentRf"(identRfAllUnits := "IdentRfHmi".unitIdentRf,   // "GetIdentRf"
                    numberOfRfReaders := "NO_OF_RF_IDENT_DEVICES",
                    IdentRfInterfaceHmi := "IdentRfInterfaceHmi");
END_REGION

REGION Network 10: Call_ MV500 Demo
   RUNG wire#powerrail
      "DemoIdentMv"()
   END_RUNG
   // the same network as SCL:
   "DemoIdentMv"();
END_REGION

REGION Network 11: Call: Diagnosticsa Ident MV
   RUNG wire#powerrail
      "InstGetIdentMv"(identMvAllUnits := "IdentMvHmi".unitIdentMv, numberOfMvReaders := "NO_OF_MV_IDENT_DEVICES", IdentMvInterfaceHmi := "IdentMvInterfaceHmi", selectedUnit =>, selectedEM =>, error =>)
   END_RUNG
   // the same network as SCL:
   "InstGetIdentMv"(identMvAllUnits := "IdentMvHmi".unitIdentMv,   // "GetIdentMv"
                    numberOfMvReaders := "NO_OF_MV_IDENT_DEVICES",
                    IdentMvInterfaceHmi := "IdentMvInterfaceHmi");
END_REGION

REGION Network 12: Call: Diagnostics Status
   RUNG wire#powerrail
      "InstProfinetDeviceDiagStatus"(devStateHmi_X1 := "PNDevDiagInterface_X1".devStateHmi, devStateHmi_X2 := "PNDevDiagInterface_X2".devStateHmi, UnitSelect := "HMI_Interface_Parameter".ProcessUnitSelect, Reset :=, DevState := "PNDevDiagStatus")
   END_RUNG
   // the same network as SCL:
   "InstProfinetDeviceDiagStatus"(devStateHmi_X1 := "PNDevDiagInterface_X1".devStateHmi,   // "LER_DiagnosticsStatus"
                           devStateHmi_X2 := "PNDevDiagInterface_X2".devStateHmi,
                           UnitSelect := "HMI_Interface_Parameter".ProcessUnitSelect,
                           DevState := "PNDevDiagStatus");
END_REGION
END_FUNCTION
